PROGRAM Combined_Vertical_Calibration
VAR
END_VAR

astAxes[AXIS_COMBINED_VERTICAL_CALIBRATION].stControl.bEnable := TRUE;
astAxes[AXIS_COMBINED_VERTICAL_CALIBRATION].stInputs.bLimitBwd := astAxes[AXIS_COMBINED_VERTICAL].stInputs.bLimitBwd;
astAxes[AXIS_COMBINED_VERTICAL_CALIBRATION].stInputs.bLimitFwd := astAxes[AXIS_COMBINED_VERTICAL].stInputs.bLimitFwd;

astAxes[AXIS_COMBINED_VERTICAL_CALIBRATION].stDescription.sAxisName := 'CALIB_Y';

END_PROGRAM

(* stored: Version 1.1.0.1, ProductVersion 3.1.4024.12
   POU Combined_Vertical_Calibration: Id {b4a07134-d384-42ed-b375-4ae5ecdec1a2}, SpecialFunc None *)
